# EPICS StreamDevice protocol: protocols/pig.proto
Terminator = LF;
ExtraInput = Ignore;

#setDDS

setDDS {
	out "dds_phase_inc 0x%x";
	in;
}
